INTERFACE I_LoadCtrl

PROPERTY bReady : BOOL
GET
END_GET
END_PROPERTY

// Show only events with minimum severety level
{attribute 'monitoring' := 'call'}
PROPERTY eTraceLevel: Global.TcEventSeverity
GET
END_GET
SET
END_SET
END_PROPERTY

PROPERTY stLoadSetpoint : ST_CtrlDataSetpoint
GET
END_GET
SET
END_SET
END_PROPERTY

PROPERTY stPowerActual : ST_CtrlDataPower
GET
END_GET
END_PROPERTY

PROPERTY stPowerMaximum : ST_CtrlDataPower
GET
END_GET
END_PROPERTY

END_INTERFACE

(* stored: Version 1.1.0.1
   Itf I_LoadCtrl: Id {86ac40be-6f7e-457b-a50f-1c0741eeb0be}
   Property bReady: Id {d85c3b98-5ee7-4ea3-bcf6-43d55bdb25a3}
   Get Get: Id {fff75793-b657-479c-a799-0000c3b98113}
   Property eTraceLevel: Id {03d013ae-a6a4-4e27-9fe6-5b041bd9a1df}
   Get Get: Id {744fcfcb-95cb-4a94-9884-31ee79ecc251}
   Set Set: Id {a50fbca3-8b01-417a-86b0-516ad9ff5cb7}
   Property stLoadSetpoint: Id {e5eefd65-9691-4c82-8abb-3737a28ac794}
   Get Get: Id {72f63399-75bb-451a-a2e3-488987d2bd2e}
   Set Set: Id {0a3ccf6c-a9a1-4a4c-9903-1aa1d27ab4b4}
   Property stPowerActual: Id {a60739b9-6ee1-440e-b842-c81015b635ad}
   Get Get: Id {0709ad5c-a181-447e-b8f7-5b72a8af5d81}
   Property stPowerMaximum: Id {48753cf6-8d8e-4257-b5b4-54483ee483a8}
   Get Get: Id {421bec78-ee1e-4ff7-a0d3-613401af118a} *)
